(*
    This function block holds all data that defines a test.
*)
FUNCTION_BLOCK FB_Test
VAR
    TestName : Tc2_System.T_MaxString;
    TestIsFinished : BOOL;
    TestIsSkipped : BOOL; // This is set to true, if test is disabled (by putting the string "disabled_" in front of the test name
    NumberOfAssertions : UINT;

    (* In which order/sequence relative to the order tests should this test be executed/evaluated.
       A value of 0 means it is not defined by TEST_ORDERED() but by un-ordered test (TEST()).
       A value <> 0 tells in which order this test will be executed/evaluated. The lower the number, the earlier it will execute. *)
    TestOrderNumber : UINT(0..GVL_Param_TcUnit.MaxNumberOfTestsForEachTestSuite); 

    (* Failure parameters. If TestIsFailed is TRUE, the other parameters will hold values as well *)
    TestIsFailed : BOOL; // Indication of whether this test has at least one failed assert
    AssertionMessage : Tc2_System.T_MaxString; // Assertion message for the first assertion in this test
    AssertionType : E_AssertionType; // Assertion type for the first assertion in this test
END_VAR

METHOD INTERNAL GetAssertionMessage : Tc2_System.T_MaxString
GetAssertionMessage := AssertionMessage;
END_METHOD

METHOD INTERNAL GetAssertionType : E_AssertionType
GetAssertionType := AssertionType;
END_METHOD

METHOD INTERNAL GetName : Tc2_System.T_MaxString;
GetName := TestName;
END_METHOD

METHOD INTERNAL GetNumberOfAssertions : UINT
GetNumberOfAssertions := NumberOfAssertions;
END_METHOD

(* Gets in which order/sequence relative to the order tests should this test be executed/evaluated. *)
METHOD INTERNAL GetTestOrder : UINT(0..GVL_Param_TcUnit.MaxNumberOfTestsForEachTestSuite);
GetTestOrder := TestOrderNumber;
END_METHOD

METHOD INTERNAL IsFailed : BOOL
IsFailed := TestIsFailed;
END_METHOD

METHOD INTERNAL IsFinished : BOOL
IsFinished := TestIsFinished;
END_METHOD

METHOD INTERNAL IsSkipped : BOOL
IsSkipped := TestIsSkipped;
END_METHOD

METHOD INTERNAL ResetTest
TestIsFinished 	:= FALSE;
TestIsSkipped	:= FALSE;
TestIsFailed	:= FALSE;
END_METHOD

(* Sets the assertion message. If one already exists, it's not overwritten as we keep the first assertion in the test *)
METHOD INTERNAL SetAssertionMessage
VAR_INPUT
    AssertMessage : Tc2_System.T_MaxString;
END_VAR
IF Tc2_Standard.LEN(STR := AssertionMessage) = 0 THEN
    AssertionMessage := AssertMessage;
END_IF
END_METHOD

(* Sets the assertion type. If one already exists, it's not overwritten as we keep the first assertion in the test *)
METHOD INTERNAL SetAssertionType
VAR_INPUT
    AssertType : E_AssertionType;
END_VAR
IF AssertionType = E_AssertionType.Type_UNDEFINED THEN
    AssertionType := AssertType;
END_IF
END_METHOD

METHOD INTERNAL SetFailed
TestIsFailed := TRUE;
END_METHOD

METHOD INTERNAL SetFinished : BOOL
TestIsFinished := TRUE;
END_METHOD

METHOD INTERNAL SetName
VAR_INPUT
    Name : Tc2_System.T_MaxString;
END_VAR
TestName := Name;
END_METHOD

METHOD INTERNAL SetNumberOfAssertions
VAR_INPUT
    NoOfAssertions : UINT;
END_VAR
NumberOfAssertions := NoOfAssertions;
END_METHOD

(* Sets the test case to skipped *)
METHOD INTERNAL SetSkipped
TestIsSkipped := TRUE;
END_METHOD

(* Sets in which order/sequence relative to the order tests should this test be executed/evaluated. *)
METHOD INTERNAL SetTestOrder
VAR_INPUT
    OrderNumber : UINT(0..GVL_Param_TcUnit.MaxNumberOfTestsForEachTestSuite);
END_VAR
TestOrderNumber := OrderNumber;
END_METHOD

END_FUNCTION_BLOCK

(* stored: Version 1.1.0.1, ProductVersion 3.1.4024.11
   POU FB_Test: Id {a51e9086-33ec-4162-acad-93a76961e893}, SpecialFunc None
   Method GetAssertionMessage: Id {273c4e89-faee-43b5-803d-428cdf75ac48}
   Method GetAssertionType: Id {cd1419c3-7b07-4183-b487-40bdbb0bbce3}
   Method GetName: Id {94757f0e-9979-49d0-ad9f-e35c823175d4}
   Method GetNumberOfAssertions: Id {0cfa1f03-0295-4f8f-bfd9-24d7b7f17e37}
   Method GetTestOrder: Id {c2cf620d-27f0-4dc3-9f43-cee6a8334a60}
   Method IsFailed: Id {e42409e3-251f-4133-8b14-3630785983d6}
   Method IsFinished: Id {813a9067-b864-4739-9c14-830160e0eabc}
   Method IsSkipped: Id {ff97feb1-1a4a-4f36-ba1d-f8483e588d4f}
   Method ResetTest: Id {e281d3d6-134a-4b52-9d17-a911235d8e0a}
   Method SetAssertionMessage: Id {05091715-93d7-47f7-9b6c-cb2511f88eb7}
   Method SetAssertionType: Id {f885f3cc-c862-4d38-9dbb-f44d7639f6a8}
   Method SetFailed: Id {b840b41b-4045-4fd9-b97d-0bf226c46fb3}
   Method SetFinished: Id {e1245d1c-be22-4d60-bc91-fe0262827234}
   Method SetName: Id {4c12f6eb-bbe4-4872-ac89-4411e2e81414}
   Method SetNumberOfAssertions: Id {94c630e9-29b9-45f4-8716-809aab6fb076}
   Method SetSkipped: Id {e9a94cad-c60d-4460-92bf-2b70cf2f46b2}
   Method SetTestOrder: Id {9154b373-5715-4bb9-b58b-0dd484b21841} *)
